// TIA Portal V17 export
// export: Created 2025-06-25T13:13:28.9414242Z, ExportSetting WithDefaults, DisplayName Totally Integrated Automation Portal, DisplayVersion V17 Update 8, DisplayName TIA Portal Openness, DisplayVersion V17 Update 8, DisplayName TIA Portal Version Control Interface, DisplayVersion V17, DisplayName STEP 7 Professional, DisplayVersion V17 Update 8, DisplayName STEP 7 Safety, DisplayVersion V17 Update 6, DisplayName WinCC Advanced, DisplayVersion V17 Update 8
TYPE "stSM522_32DQ_I"
// stored: IsFailsafeCompliant false
   STRUCT
      DQ00_ok : Bool;
      DQ01_ok : Bool;
      DQ02_ok : Bool;
      DQ03_ok : Bool;
      DQ04_ok : Bool;
      DQ05_ok : Bool;
      DQ06_ok : Bool;
      DQ07_ok : Bool;
      DQ08_ok : Bool;
      DQ09_ok : Bool;
      DQ10_ok : Bool;
      DQ11_ok : Bool;
      DQ12_ok : Bool;
      DQ13_ok : Bool;
      DQ14_ok : Bool;
      DQ15_ok : Bool;
      DQ16_ok : Bool;
      DQ17_ok : Bool;
      DQ18_ok : Bool;
      DQ19_ok : Bool;
      DQ20_ok : Bool;
      DQ21_ok : Bool;
      DQ22_ok : Bool;
      DQ23_ok : Bool;
      DQ24_ok : Bool;
      DQ25_ok : Bool;
      DQ26_ok : Bool;
      DQ27_ok : Bool;
      DQ28_ok : Bool;
      DQ29_ok : Bool;
      DQ30_ok : Bool;
      DQ31_ok : Bool;
   END_STRUCT;
END_TYPE
